Fanuc KAREL source: remote_position.kl

PROGRAM remoteposition
%COMMENT = ' Remote Position'
%NOLOCKGROUP
%NOBUSYLAMP

CONST
	PR_XYZWPR = 41

VAR
	rf_ :FILE
	STATUS: INTEGER
	current_pos: XYZWPR

BEGIN

	$GROUP[1].$UTOOL = $MNUTOOL[1,1] --uTool 1
	$GROUP[1].$UFRAME = $MNUFRAME[1,1] --uFrame 1
	current_pos = CURPOS(0,0)

	OPEN FILE rf_ ('RW', 'RD:RESPONSE.HTM')
	STATUS = IO_STATUS(rf_)
	IF (STATUS <> 0) THEN
		WRITE rf_ ( '{"result":"failed", "reason":',STATUS,'}')
	ELSE
		WRITE rf_ (  '{"result":"success"',
					', "x":', current_pos.x,
					', "y":', current_pos.y,
					', "z":', current_pos.z,
					', "w":', current_pos.w,
					', "p":', current_pos.p,
					', "r":', current_pos.r,
					'}', CR)
	ENDIF
	CLOSE FILE rf_
END remoteposition
